{attribute 'GeneratedUsingTerminal: EK1100-0000-0018'}
{attribute addProperty BoxType "EK1100-0000-0018"}
{attribute addProperty Id "Beckhoff_EL68xxEK1122Beckhoff_EL68xxEK1122_4A27306B2A_0001_EL6851_0000_0017EL6851_A971184B539A_0002_EL6851_0000_0018EL6851_A971184B539A_0003_EL6851_0000_0019EL6851_A971184B539A_0004_EL6851_0000_0020EL6851_A971184B539A_0005_EL6851_0000_0021EL6851_A971184B539A_0006_EL6851_0010_0016EL6851_CAB27A3184A_0007_EL6851_0010_0017EL6851_CAB27A3184A_0008_EL6851_0010_0018EL6851_CAB27A3184A_0009_EL6851_0010_0019EL6851_CAB27A3184A_0010_EL6861_0000_0016EL6861_D3CF2867282A_0011_EL6861_0000_0017EL6861_D3CF2867282"}
{attribute addProperty CRC "1986454992"}
{attribute addProperty Size "3597"}
TYPE Beckhoff_EL68xx_7666E5D0 EXTENDS EK1100_AB5A9467 :
STRUCT
	{attribute addProperty Name "Beckhoff_EL68xxEK1122"}
	Beckhoff_EL68xxEK1122 : Beckhoff_EL68xxEK1122_4A27306B;
	{attribute addProperty Name "A_0001_EL6851_0000_0017"}
	A_0001_EL6851_0000_0017 : EL6851_A971184B;
	{attribute addProperty Name "A_0002_EL6851_0000_0018"}
	A_0002_EL6851_0000_0018 : EL6851_A971184B;
	{attribute addProperty Name "A_0003_EL6851_0000_0019"}
	A_0003_EL6851_0000_0019 : EL6851_A971184B;
	{attribute addProperty Name "A_0004_EL6851_0000_0020"}
	A_0004_EL6851_0000_0020 : EL6851_A971184B;
	{attribute addProperty Name "A_0005_EL6851_0000_0021"}
	A_0005_EL6851_0000_0021 : EL6851_A971184B;
	{attribute addProperty Name "A_0006_EL6851_0010_0016"}
	A_0006_EL6851_0010_0016 : EL6851_CAB27A31;
	{attribute addProperty Name "A_0007_EL6851_0010_0017"}
	A_0007_EL6851_0010_0017 : EL6851_CAB27A31;
	{attribute addProperty Name "A_0008_EL6851_0010_0018"}
	A_0008_EL6851_0010_0018 : EL6851_CAB27A31;
	{attribute addProperty Name "A_0009_EL6851_0010_0019"}
	A_0009_EL6851_0010_0019 : EL6851_CAB27A31;
	{attribute addProperty Name "A_0010_EL6861_0000_0016"}
	A_0010_EL6861_0000_0016 : EL6861_D3CF2867;
	{attribute addProperty Name "A_0011_EL6861_0000_0017"}
	A_0011_EL6861_0000_0017 : EL6861_D3CF2867;
END_STRUCT
END_TYPE

(* stored: Version 1.2.0.0, ProductVersion 3.1.4024.9
   DUT Beckhoff_EL68xx_7666E5D0: Id {585e9a77-cc83-4b40-b46a-c3775d2ee943} *)
